{attribute addProperty BoxType "EL2262-0000-0001"}
{attribute addProperty Id "Cycle_CounterAT %Q*UINT162"}
{attribute addProperty CRC "1213625600"}
{attribute addProperty SizeInBites "16"}
{attribute addProperty SizeInBytes "2"}
TYPE CycCount1_48567500 :
STRUCT
	{attribute addProperty Name "Cycle_Counter"}
	Cycle_Counter AT %Q* : UINT;
END_STRUCT
END_TYPE

(* stored: Version 1.2.0.0, ProductVersion 3.1.4024.9
   DUT CycCount1_48567500: Id {28f96adc-5fb3-4e5c-bd03-00a95939e257} *)
